FUNCTION_BLOCK FB_PalletStation EXTENDS FB_Module IMPLEMENTS I_GantryPallet
VAR_INPUT
	Axis				: REFERENCE TO AXIS_REF;
	ipGantry1			: I_GantryPallet;
	ipGantry2			: I_GantryPallet;
	cmd					: E_PalletStationCommand := E_PalletStationCommand.None;
	
	inpPalletRecord		: REFERENCE TO ARRAY[0..100] OF ST_PalletRecord;
	inpActiveRecord		: REFERENCE TO DINT;	
	inpSim				: BOOL := TRUE;
	inpPalletPresent	AT %I* : BOOL;
END_VAR
VAR_OUTPUT
	stsState			: E_PalletStationState := E_PalletStationState.Idle;
	stsCurrentStep		: DINT;
END_VAR
VAR
	//Devices
	Conveyor			: FB_Axis;
	PalletStop			: FB_Actuator;
	RFID				: FB_RFID;
	
	DepartureTimer		: TON;
	DepartureDelayTime	: TIME := T#3S;
	PP_DepartSimTimer	: TON;
	PP_ArriveSimTimer	: TON;
	
	rtStarting			: R_TRIG;
	rtStopping			: R_TRIG;
	rtHoming			: R_TRIG;
	rtPalletPresent		: R_TRIG;

	i					: DINT;	
	j					: DINT;
	Gantry1Clear		: BOOL;
	Gantry2Clear		: BOOL;
END_VAR
VAR CONSTANT
	NULL_RECORD			: ARRAY[1..100] OF STRING;
END_VAR

Map();
Status();
StateMachine();

METHOD Aborting : BOOL
VAR_INPUT
END_VAR
Conveyor.cmd := E_AxisCommand.Stop;
stsCurrentStep := 0;
END_METHOD

METHOD Homing : BOOL
VAR_INPUT
END_VAR
CASE stsCurrentStep OF
	4000: //Clear RFID and active record
		RFID.cmd := E_RFIDCommand.Clear;
		inpActiveRecord := 0;
		IF RFID.stsCurrentID = '' THEN
			stsCurrentStep := 4010;
		END_IF
	4010: //Extend pallet stop
		PalletStop.cmd := E_ActuatorCommand.Work;
		IF PalletStop.stsState = E_ActuatorState.AtWork THEN
			stsCurrentStep := 4020;
		END_IF
	4020: //Stop conveyor
		Conveyor.cmd := E_AxisCommand.Stop;
		IF Conveyor.stsVelocity = 0 THEN
			stsCurrentStep := 0;
		END_IF
END_CASE
END_METHOD

METHOD Map : BOOL
VAR_INPUT
END_VAR
Conveyor(Axis := Axis);
PalletStop();
RFID();

DepartureTimer(IN := stsCurrentStep = 3050 AND NOT inpPalletPresent, PT := DepartureDelayTime);

Gantry1Clear := ipGantry1.PalletReady;
Gantry2Clear := ipGantry2.PalletReady;
END_METHOD

{warning 'add property implementation'}
PROPERTY PalletReady : BOOL
GET
PalletReady := inpPalletPresent AND Gantry1Clear AND Gantry2Clear AND PalletStop.stsState = E_ActuatorState.AtWork;
END_GET
END_PROPERTY

METHOD Running : BOOL
VAR_INPUT
END_VAR
CASE stsCurrentStep OF
	3000: //Read RFID
		RFID.cmd := E_RFIDCommand.Read;
		IF RFID.stsCurrentID <> '' THEN
			stsCurrentStep := 3010;
		END_IF
	3010: //Clear associated data
		FOR i := 1 TO 100 DO
			IF inpPalletRecord[i].ID = RFID.stsCurrentID THEN
				inpPalletRecord[i].Data := NULL_RECORD;
				inpActiveRecord := i;
				stsCurrentStep := 3020;
			END_IF
		END_FOR
	3020: //Wait for all 12 records to populate
		IF (inpPalletRecord[inpActiveRecord].Data[1] <> '' AND
			inpPalletRecord[inpActiveRecord].Data[2] <> '' AND
			inpPalletRecord[inpActiveRecord].Data[3] <> '' AND
			inpPalletRecord[inpActiveRecord].Data[4] <> '' AND
			inpPalletRecord[inpActiveRecord].Data[5] <> '' AND
			inpPalletRecord[inpActiveRecord].Data[6] <> '' AND
			inpPalletRecord[inpActiveRecord].Data[7] <> '' AND
			inpPalletRecord[inpActiveRecord].Data[8] <> '' AND
			inpPalletRecord[inpActiveRecord].Data[9] <> '' AND
			inpPalletRecord[inpActiveRecord].Data[10] <> '' AND
			inpPalletRecord[inpActiveRecord].Data[11] <> '' AND
			inpPalletRecord[inpActiveRecord].Data[12] <> '')
		THEN
			inpActiveRecord := 0;
			stsCurrentStep := 3030;
		END_IF
	3030: //Wait for gantries to clear station
		IF Gantry1Clear AND Gantry2Clear THEN
			stsCurrentStep := 3040;
		END_IF
	3040: //Release pallet
		PalletStop.cmd := E_ActuatorCommand.Home;
		IF PalletStop.stsState = E_ActuatorState.AtHome THEN
			stsCurrentStep := 3050;
		END_IF
	3050: //Wait for pallet to leave
		IF DepartureTimer.Q THEN
			stsCurrentStep := 3060;
		END_IF
	3060: //Extend pallet stop
		PalletStop.cmd := E_ActuatorCommand.Work;
		IF PalletStop.stsState = E_ActuatorState.AtWork THEN
			stsCurrentStep := 3070;
		END_IF
	3070: //Clear RFID
		RFID.cmd := E_RFIDCommand.Clear;
		IF RFID.stsCurrentID = '' THEN
			stsCurrentStep := 0;
		END_IF
END_CASE
END_METHOD

METHOD Simulate : BOOL
VAR_INPUT
END_VAR
PP_DepartSimTimer(IN := stsCurrentStep = 3050, PT := T#5S);
inpPalletPresent R= PP_DepartSimTimer.Q;

PP_ArriveSimTimer(IN := stsState = E_PalletStationState.Running AND NOT inpPalletPresent, PT := T#10S);
inpPalletPresent S= PP_ArriveSimTimer.Q;
END_METHOD

METHOD Starting : BOOL
VAR_INPUT
END_VAR
CASE stsCurrentStep OF
	1000: //Clear RFID
		RFID.cmd := E_RFIDCommand.Clear;
		IF RFID.stsCurrentID = '' THEN
			stsCurrentStep := 1010;
		END_IF
	1010: //Extend pallet stop
		PalletStop.cmd := E_ActuatorCommand.Work;
		IF PalletStop.stsState = E_ActuatorState.AtWork THEN
			stsCurrentStep := 1020;
		END_IF
	1020: //Turn on conveyor
		Conveyor.cmd := E_AxisCommand.TurnOn;
		IF Conveyor.stsState = E_AxisState.Ready THEN
			stsCurrentStep := 1030;
		END_IF
	1030: //Run conveyor at 100 mm/s (arbitrary value for project)
		Conveyor.inpVelocity := 100;
		Conveyor.cmd := E_AxisCommand.ExecuteMoveVel;
		IF Conveyor.stsVelocity > 0 THEN
			stsCurrentStep := 0;
		END_IF
END_CASE
END_METHOD

METHOD StateMachine : BOOL
VAR_INPUT
END_VAR
IF inpSim THEN
	Simulate();
END_IF

CASE stsState OF
	E_PalletStationState.Idle: //Station idle and ready for command
		IF cmd = E_PalletStationCommand.Start THEN
			stsState := E_PalletStationState.Starting;
		ELSIF cmd = E_PalletStationCommand.Home THEN
			stsState := E_PalletStationState.Homing;
		END_IF
	E_PalletStationState.Homing: //Return station to home state
		Homing();
		IF stsCurrentStep = 0 AND PalletStop.stsState = E_ActuatorState.AtWork THEN
			stsState := E_PalletStationState.Idle;
		END_IF
	E_PalletStationState.Starting: //Start conveyor and ready to process
		Starting();
		IF stsCurrentStep = 0 AND Conveyor.stsVelocity > 0 AND PalletStop.stsState = E_ActuatorState.AtWork THEN
			stsState := E_PalletStationState.Running;
		END_IF
	E_PalletStationState.Running: //Station is running and ready to receive pallet
		Running();
		IF cmd = E_PalletStationCommand.Stop THEN
			Stopping();
			stsState := E_PalletStationState.Stopping;
		END_IF
	E_PalletStationState.Stopping: //Station is stopping
		Stopping();
		IF stsCurrentStep = 0 AND Conveyor.stsVelocity = 0 AND PalletStop.stsState = E_ActuatorState.AtWork THEN
			stsState := E_PalletStationState.Idle;
		END_IF
	E_PalletStationState.Aborting: //Abort all station activity
		Aborting();
		IF stsCurrentStep = 0 AND Conveyor.stsVelocity = 0 THEN
			stsState := E_PalletStationState.Idle;
		END_IF		
END_CASE

IF cmd = E_PalletStationCommand.Abort THEN
	stsState := E_PalletStationState.Aborting;
END_IF

cmd := E_PalletStationCommand.None;
END_METHOD

METHOD Status : BOOL
VAR_INPUT
END_VAR
//State transition one shots
rtStarting(CLK := stsState = E_PalletStationState.Starting);
IF rtStarting.Q THEN
	stsCurrentStep := 1000;
END_IF

rtStopping(CLK := stsState = E_PalletStationState.Stopping);
IF rtStopping.Q THEN
	stsCurrentStep := 2000;
END_IF

rtHoming(CLK := stsState = E_PalletStationState.Homing);
IF rtHoming.Q THEN
	stsCurrentStep := 4000;
END_IF

rtPalletPresent(CLK := inpPalletPresent AND stsState <> E_PalletStationState.Homing AND stsCurrentStep = 0);
IF rtPalletPresent.Q THEN
	stsCurrentStep := 3000;
END_IF
END_METHOD

METHOD Stopping : BOOL
VAR_INPUT
END_VAR

VAR
	END_IFCASE: INT;
END_VAR
CASE stsCurrentStep OF
	2000: //Clear RFID
		RFID.cmd := E_RFIDCommand.Clear;
		IF RFID.stsCurrentID = '' THEN
			stsCurrentStep := 2010;
		END_IF
	2010: //Extend pallet stop
		PalletStop.cmd := E_ActuatorCommand.Work;
		IF PalletStop.stsState = E_ActuatorState.AtWork THEN
			stsCurrentStep := 2020;
		END_IF
	2020: //Stop conveyor
		Conveyor.cmd := E_AxisCommand.Stop;
		IF Conveyor.stsVelocity = 0 THEN
			stsCurrentStep := 0;
		END_IF
END_CASE
END_METHOD

END_FUNCTION_BLOCK

(* stored: Version 1.1.0.1, ProductVersion 3.1.4024.4
   POU FB_PalletStation: Id {5588170d-2109-4a73-9f01-47cd58a5f839}, SpecialFunc None
   Method Aborting: Id {307137c9-b7bf-4c89-9bbf-10b9561aedc3}
   Method Homing: Id {a84e6e5b-e2c2-4d0d-a14c-11d6c2c85e32}
   Method Map: Id {1d064eb5-c2a7-4c82-a039-8d10d4723f06}
   Property PalletReady: Id {7eee9fc2-7b02-4a0e-bf54-ce2641ef3ed1}
   Get Get: Id {b44be487-40dc-4043-9af0-370abe2c1740}
   Method Running: Id {918a504f-8e24-4f70-a661-e59c95146542}
   Method Simulate: Id {d72fc5d7-22e7-4fb4-be7a-6f1ca20d6a35}
   Method Starting: Id {212b0d79-875f-4a91-bcfc-7910befee0c7}
   Method StateMachine: Id {25eb7868-e248-4632-b391-42aa626a08bc}
   Method Status: Id {e3cb56af-697a-48ef-8b91-167b8b67fb5d}
   Method Stopping: Id {1cb79882-1e69-4491-abea-c356ba24106f} *)
